FUNCTION_BLOCK FB_Module EXTENDS FB_Element IMPLEMENTS I_Module
VAR_INPUT
END_VAR
VAR_OUTPUT
END_VAR
VAR
	{attribute 'OPC.UA.DA' := '1'}
	{attribute 'OPC.UA.DA.Access' := '2'}
	eMode:							E_Mode;							// Current mode
		{attribute 'OPC.UA.DA' := '1'}
	{attribute 'OPC.UA.DA.Access' := '1'}
	eModeRequest:					E_Mode:= E_Mode.Automatic;		// Requested mode
	{attribute 'hide'}
	eModePrevious:					E_Mode;							// Previous mode
	
	fbLogging:					FB_LoggingProvider;
	fbLogger:					FB_Logger<20>;
	
	fbLevel1:					FB_Level;
	fbLevel2:					FB_Level;
END_VAR

// https://peterzerlauth.com/
SUPER^();

fbLogger();

fbLevel1();
fbLevel2();

// Detect mode changes
IF eModeRequest <> E_Mode.Undefined THEN
	IF eMode <> eModeRequest THEN
		eModePrevious:= eMode;
		eMode:= eModeRequest;
		M_OnMode(eMode, eModePrevious);
	END_IF
END_IF
eModeRequest:= E_Mode.Undefined;

METHOD PROTECTED M_Aborting : BOOL (* Return*)
M_Aborting:= 	fbLevel2.M_Request(E_Request.Abort) AND
				fbLevel1.M_Request(E_Request.Abort);
END_METHOD

METHOD PROTECTED M_Idle : BOOL (* Return*)
fbLogging.M_Add(fbLogger);


P_Event.P_Logger:= fbLogging;
fbLevel2.P_Event.P_Logger:= fbLogging;
fbLevel1.P_Event.P_Logger:= fbLogging;

fbLevel2.P_Event.P_Observer.M_Attach(THIS^);
fbLevel1.P_Event.P_Observer.M_Attach(THIS^);

fbLevel2.M_Attach(fbLevel1);

fbEvent.fbObserver.M_Attach(fbLevel1);
END_METHOD

{attribute 'TcRpcEnable':='1'}
METHOD PUBLIC M_Mode : BOOL
VAR_INPUT
	eMode:		E_Mode;
END_VAR
IF THIS^.eMode = eMode THEN
	M_Mode:= TRUE;
ELSE
	eModeRequest:= eMode;	
END_IF
END_METHOD

METHOD PROTECTED M_OnMode
VAR_INPUT
	eMode:							E_Mode;						// Current mode
	eModePrevious:					E_Mode;						// Previous mode	
END_VAR
CASE eMode OF
	E_Mode.Semiauto, E_Mode.Automatic:
		IF eModePrevious = E_Mode.Manual THEN
			fbEvent.M_AddSTRING(TO_STRING(eModePrevious));
			fbEvent.M_AddSTRING(TO_STRING(eMode));
			fbEvent.M_Fatal('Module mode changed form %s to %s', 1002);
		END_IF
	E_Mode.Manual:
		;
END_CASE
END_METHOD

METHOD PROTECTED M_Resetting : BOOL (* Return*)
M_Resetting:= 	fbLevel2.M_Request(E_Request.Reset) AND
				fbLevel1.M_Request(E_Request.Reset);
END_METHOD

METHOD PROTECTED M_Starting : BOOL
VAR_INPUT
END_VAR
M_Starting:= 	fbLevel1.M_Request(E_Request.Start) AND_THEN fbLevel2.M_Request(E_Request.Start);
END_METHOD

METHOD PROTECTED M_Stopping : BOOL (* Return state complete*)
M_Stopping:= 	fbLevel2.M_Request(E_Request.Stop) AND
				fbLevel1.M_Request(E_Request.Stop);
END_METHOD

PROPERTY PUBLIC P_Mode : E_Mode
GET
P_Mode:= eMode;
END_GET
END_PROPERTY

END_FUNCTION_BLOCK

(* stored: Version 1.1.0.1
   POU FB_Module: Id {0d3fc497-598e-0d21-1617-ce19be6391a0}, SpecialFunc None
   Method M_Aborting: Id {1929bb83-c65f-09d2-2a22-b68806b0f4ac}
   Method M_Idle: Id {53713e89-9f8a-0ca1-3503-bec2867bc268}
   Method M_Mode: Id {8661b760-0fa5-007a-151c-7fe805544fbb}
   Method M_OnMode: Id {549d817a-659a-0f3e-10ea-6f23f3ce8adf}
   Method M_Resetting: Id {dd412173-49e2-0d05-1622-bbd0077f06b6}
   Method M_Starting: Id {6fe2f334-328e-0cdd-0d07-134e9af3083f}
   Method M_Stopping: Id {36c858d8-accc-01ae-0f5b-a1e3f137f544}
   Property P_Mode: Id {a773e62d-20bd-0c96-369b-0f3305d57073}
   Get Get: Id {0b059178-babf-076f-2ccc-02e13582bfc7} *)
